// SIMATIC STEP 7 (V5.x) project GATE_RS
// program: S7 Program(1)

SYMBOL_TABLE
"GATE_RS"	FB 139	FB 139
END_SYMBOL_TABLE

FUNCTION_BLOCK "GATE_RS"	// FB 139
AUTHOR : ETSystem
VERSION : 0.1
VAR_INPUT
  MAN : BOOL ;
  COMMON_FAULT : BOOL ;
  AUTO : BOOL ;
  PAZ_FAULT : BOOL ;
END_VAR
VAR_OUTPUT
  QMAN : BOOL ;
  QAUTO : BOOL ;
END_VAR
BEGIN
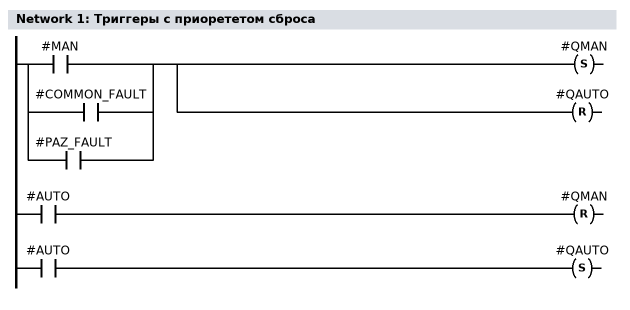
NETWORK
TITLE = Триггеры с приорететом сброса
      O     #MAN;
      O     #COMMON_FAULT;
      O     #PAZ_FAULT;
      =     L 0.0;
      A     L 0.0;
      S     #QMAN;
      A     #AUTO;
      R     #QMAN;
      NOP   0;
      A     #AUTO;
      S     #QAUTO;
      A     L 0.0;
      R     #QAUTO;
      NOP   0;
END_FUNCTION_BLOCK

ORGANIZATION_BLOCK OB 1
TITLE = "Main Program Sweep (Cycle)"
VERSION : 0.1
VAR_TEMP
  OB1_EV_CLASS : BYTE ;	//Bits 0-3 = 1 (Coming event), Bits 4-7 = 1 (Event class 1)
  OB1_SCAN_1 : BYTE ;	//1 (Cold restart scan 1 of OB 1), 3 (Scan 2-n of OB 1)
  OB1_PRIORITY : BYTE ;	//Priority of OB Execution
  OB1_OB_NUMBR : BYTE ;	//1 (Organization block 1, OB1)
  OB1_RESERVED_1 : BYTE ;	//Reserved for system
  OB1_RESERVED_2 : BYTE ;	//Reserved for system
  OB1_PREV_CYCLE : INT ;	//Cycle time of previous OB1 scan (milliseconds)
  OB1_MIN_CYCLE : INT ;	//Minimum cycle time of OB1 (milliseconds)
  OB1_MAX_CYCLE : INT ;	//Maximum cycle time of OB1 (milliseconds)
  OB1_DATE_TIME : DATE_AND_TIME ;	//Date and time OB1 started
END_VAR
BEGIN
// (block stored without names or comments; labels and parameter names are numbered)
END_ORGANIZATION_BLOCK
